(* PLC project KinIn_v3.project, CODESYS CODESYS V3.5 SP19 *)
(* stored: creationDateTime 2025-01-20T16:26:01.6267276, modificationDateTime 2025-01-20T16:17:39.6822999 *)

FUNCTION_BLOCK so3ToAngularVelocity
  VAR_INPUT
    so3mat : ARRAY[1..3, 1..3] OF REAL;  (* so3x3 *)
  END_VAR
  VAR_OUTPUT
    omg : ARRAY[1..3] OF REAL;  (* SO3x3 *)
  END_VAR

            omg[1]:=so3mat[3, 2];
omg[2]:=so3mat[1, 3];
omg[3]:=so3mat[2, 1];


          
END_FUNCTION_BLOCK
